FUNCTION_BLOCK "Syntax_MissingAssignmentSemicolon"
{ S7_Optimized_Access := 'TRUE' }
VERSION : 0.1

VAR
    a        : Int := 1;
    b        : Int := 2;
    result   : Int := 0;
    flag     : Bool := TRUE;
    i        : Int := 0;
    values   : Array[0..9] of Int;
END_VAR
BEGIN
    #result := #a + #b
    // EXPECT: error[syntax.missing-semicolon] SYN-STMT-001
    #result := 123;
    // RECOVERY: this statement should still be parsed

END_FUNCTION_BLOCK
